TYPE "Prg_Header"
VERSION : 0.1
// Block: Prg_Header
   STRUCT
      PrgNo : DInt;
      PrgName : "String[30]";
   END_STRUCT;

END_TYPE
